FUNCTION_BLOCK TcEventClassArguments IMPLEMENTS I_EventArguments
VAR
	pArgumentEvent : POINTER TO FB_TcAlarm;
END_VAR

METHOD AddString : I_EventArguments
VAR_INPUT
	Argument : STRING;
END_VAR
IF pArgumentEvent <> 0 THEN
	pArgumentEvent^.ipArguments.AddString(Argument);
END_IF

AddString := THIS^;
END_METHOD

METHOD Clear : I_EventArguments
IF pArgumentEvent <> 0 THEN
	pArgumentEvent^.ipArguments.Clear();
END_IF

Clear := THIS^;
END_METHOD

PROPERTY Event : POINTER TO FB_TcAlarm
SET
pArgumentEvent := Event;
END_SET
END_PROPERTY

END_FUNCTION_BLOCK

(* stored: Version 1.1.0.1, ProductVersion 3.1.4026.18
   POU TcEventClassArguments: Id {4da6bc0f-f7b2-48c4-b813-e40d79558b62}, SpecialFunc None
   Method AddString: Id {8a6fa489-eeec-40ff-b2d2-3feb0d4ce074}
   Method Clear: Id {506b08da-9af2-47ec-8146-ff18e19be2d9}
   Property Event: Id {e7942ebe-6665-4923-ad58-88e5c7dffa82}
   Set Set: Id {0ff0532c-c9e0-4841-8b6f-67b32221ed3b} *)
